// TIA Portal V19 export
TYPE "stParamManuFerRobotic"
   STRUCT
      "#OutToSlave.ManualSandingPaperParam.nSetForceTarget    #OutToSlave.ManualSandingPaperParam.nSetForceZero    #OutToSlave.ManualSa" : Bool;
   END_STRUCT;
END_TYPE
